PROGRAM EventLog


VAR
	WriteTest		:	BOOL;
	fbOpenFile 		: FB_Fileopen;
	fbWriteFile		: FB_FilePuts;
	fbCloseFile 	: FB_FileClose;
	fbRenameFile	: FB_FileRename;
	fbDeleteFile	: FB_FileDelete;
	fbFileInfo		:	FB_EnumFindFileEntry;
	stFiledata		:	ST_FindFileEntry;
	FileOpenDone		:	F_TRIG;
	FileWriteDone		:	F_TRIG;
	FileCloseDone		:	F_TRIG;
	FileRenameDone		:	F_TRIG;
	FileDeleteDone		:	F_TRIG;
	FileInfoDone		:	F_TRIG;
	FileSize			:	ULINT;
	FileCounter			:	INT;
	Filehandle 			: UINT;
	
	bForceWrite 			:	BOOL;	//immediately flush out buffer on shutdown
	bEMstopWrite			:	BOOL;	//Flush out after EMStop, but give some time for final logs to come in 
	tonEMstopDelay			:	TON;
	tonGeneralWriteDelay	:	Ton;
	FileActionDelay			:	TON := (PT := T#30MS);

	MemoryBuffer	:	FB_StringRingBuffer;
	DataBuffer		:	ARRAY[0..100000] OF BYTE; //100kb to start
	WriteString	:	t_MAXSTRING;

	
	
	Stop_logging	:	Bool;
	
END_VAR

VAR_IN_OUT CONSTANT
	STParams : ST_EventLoggerParams;
END_VAR

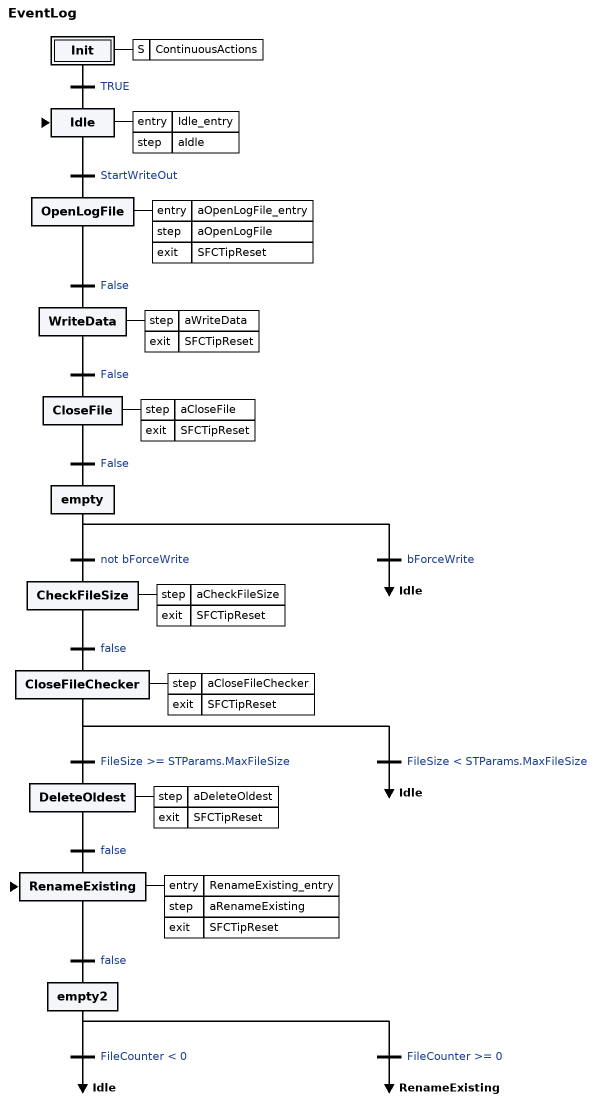
INITIAL_STEP Init:
    ContinuousActions(S);
END_STEP
TRANSITION FROM Init TO Idle
    := TRUE;
END_TRANSITION
STEP Idle:
    Idle_entry(P1);  // entry action
    aIdle(N);  // step action
END_STEP
TRANSITION FROM Idle TO OpenLogFile
    := StartWriteOut;
END_TRANSITION
// macro Writeout begins
STEP OpenLogFile:
    aOpenLogFile_entry(P1);  // entry action
    aOpenLogFile(N);  // step action
    SFCTipReset(P0);  // exit action
END_STEP
TRANSITION FROM OpenLogFile TO WriteData
    := False;
END_TRANSITION
STEP WriteData:
    aWriteData(N);  // step action
    SFCTipReset(P0);  // exit action
END_STEP
TRANSITION FROM WriteData TO CloseFile
    := False;
END_TRANSITION
STEP CloseFile:
    aCloseFile(N);  // step action
    SFCTipReset(P0);  // exit action
END_STEP
TRANSITION FROM CloseFile TO empty
    := False;
END_TRANSITION
STEP empty:
END_STEP
TRANSITION FROM empty TO CheckFileSize
    := not bForceWrite;
END_TRANSITION
TRANSITION FROM empty TO Idle
    := bForceWrite;
END_TRANSITION
// macro LogRotate begins
STEP CheckFileSize:
    aCheckFileSize(N);  // step action
    SFCTipReset(P0);  // exit action
END_STEP
TRANSITION FROM CheckFileSize TO CloseFileChecker
    := false;
END_TRANSITION
STEP CloseFileChecker:
    aCloseFileChecker(N);  // step action
    SFCTipReset(P0);  // exit action
END_STEP
TRANSITION FROM CloseFileChecker TO DeleteOldest
    := FileSize >= STParams.MaxFileSize;
END_TRANSITION
STEP DeleteOldest:
    aDeleteOldest(N);  // step action
    SFCTipReset(P0);  // exit action
END_STEP
TRANSITION FROM DeleteOldest TO RenameExisting
    := false;
END_TRANSITION
STEP RenameExisting:
    RenameExisting_entry(P1);  // entry action
    aRenameExisting(N);  // step action
    SFCTipReset(P0);  // exit action
END_STEP
TRANSITION FROM RenameExisting TO empty2
    := false;
END_TRANSITION
STEP empty2:
END_STEP
TRANSITION FROM empty2 TO Idle
    := FileCounter < 0;
END_TRANSITION
TRANSITION FROM empty2 TO RenameExisting
    := FileCounter >= 0;
END_TRANSITION
TRANSITION FROM CloseFileChecker TO Idle
    := FileSize < STParams.MaxFileSize;
END_TRANSITION

ACTION aCheckFileSize:


FileInfoDone(clk := fbFileInfo.bbusy);
FileActionDelay(in:= NOT (fbFileInfo.bbusy OR FileInfoDone.Q));

fbFileInfo(sPathname:= Stparams.LogFileName,
		bExecute := FileActionDelay.Q,
		eCMD := eEnumCmd_First,
		tTimeout := T#100MS);


IF FileInfoDone.q THEN
	FileSize := 0;
	IF NOT fbFileInfo.bError THEN
		IF NOT fbfileInfo.bEOE THEN
			stFiledata := fbFileinfo.stFindFile;
			FileSize := ULARGE_TO_ULINT(stFiledata.fileSize);
		END_IF
	END_IF
	SFCTip := TRUE;
END_IF
END_ACTION

ACTION aCloseFile:

FileCloseDone(clk := fbCloseFile.bbusy);

FileActionDelay(in := NOT (fbCloseFile.bbusy OR FileCloseDone.Q));


fbCloseFile(Hfile := FileHandle,
		bExecute   := FileActionDelay.q,
    	tTimeout   := T#100MS);


IF FileCloseDone.q THEN
	IF NOT fbCloseFile.bError THEN
		filehandle := 0;
		SFCTip := TRUE;
	END_IF
END_IF
END_ACTION

ACTION aCloseFileChecker:


FileInfoDone(clk := fbFileInfo.bbusy);
FileActionDelay(in:= not (fbFileInfo.bbusy OR FileInfoDone.Q));

fbFileInfo(sPathname:= Stparams.LogFileName,
		bExecute := FileActionDelay.Q,
		eCMD := eEnumCmd_Abort,
		tTimeout := T#100MS);


IF FileInfoDone.q THEN
	FileSize := 0;
	IF NOT fbFileInfo.bError THEN
		SFCTip := TRUE;
	END_IF
END_IF
END_ACTION

METHOD AddEvent : BOOL
VAR_INPUT
	LogMessage	:	STRING;
END_VAR
IF NOT Stop_logging THEN	
	MemoryBuffer.A_AddTail(putValue := LogMessage);
end_if
END_METHOD

ACTION aDeleteOldest:

FileDeleteDone(clk := fbDeleteFile.bbusy);
FileActionDelay(in:=NOT (fbDeleteFile.bbusy OR FileDeleteDone.Q));
	
fbDeleteFile(sPathname:= concat(concat(Stparams.LogFileName, '.'),TO_STRING(stparams.MaxFileCount-1)),
		bExecute := FileActionDelay.q,
		tTimeout := T#100MS);


IF FileDeleteDone.q THEN
	//could end in error if file doesn't exist. This is fine.
	FileCounter := stparams.MaxFileCount-2;
	SFCTip := TRUE;
END_IF
END_ACTION

ACTION aIdle:
tonGeneralWriteDelay.IN := true;
END_ACTION

ACTION aOpenLogFile:
bEMStopWrite := FALSE;
tonGeneralWriteDelay.IN := FALSE;
FileOpenDone(clk := fbOpenFile.bbusy);

FileActionDelay(in := NOT (fbOpenFile.bbusy OR FileOpenDone.Q));

fbOpenFile(sPathName := Stparams.LogFileName,
		nMode := FOPEN_MODEAPPEND OR FOPEN_MODETEXT,
		bExecute   :=  FileActionDelay.Q,
    	tTimeout   := T#100MS);


IF FileOpenDone.q THEN
	FileHandle := fbOpenFile.hFile;
	IF FileHandle <> 0 THEN
		MemoryBuffer.A_RemoveHead(getValue => WriteString);
		SFCTip := TRUE;
	END_IF
END_IF
END_ACTION

ACTION aOpenLogFile_entry:

END_ACTION

ACTION aRenameExisting:

FileRenameDone(clk := fbRenameFile.bbusy);
FileActionDelay(in:= NOT (fbDeleteFile.bbusy OR FileDeleteDone.Q));

fbRenameFile(
		bExecute := FileActionDelay.Q,
		tTimeout := T#100MS);


IF FileRenameDone.q THEN
	//could end in error if file doesn't exist. This is fine.
	FileCounter := FileCounter-1;
	SFCTip := TRUE;
END_IF
END_ACTION

ACTION aWriteData:

//add entry action with initial Writestring fill
filehandle;

FileWriteDone(clk := fbWriteFile.bbusy);

FileActionDelay(in := NOT (fbWriteFile.bbusy OR FileWriteDone.Q));

fbWriteFile(hfile := filehandle,
			sLine := WriteString,
			BExecute := FileActionDelay.Q,
			tTimeout := T#500MS);


IF FileWriteDone.q THEN
	IF MemoryBuffer.nCount > 0 THEN //Still data present, continue writing
		MemoryBuffer.A_RemoveHead(getValue => WriteString);
	ELSE //file not opened, back to start?
		SFCTip := TRUE;
	END_IF
END_IF
END_ACTION

ACTION ContinuousActions:
MemoryBuffer(bOverwrite := TRUE, pBuffer := ADR(DataBuffer), cbBuffer := SIZEOF(DataBuffer));
tonEMstopDelay(in := bEMstopWrite, pt:= stparams.EMstopWriteDelay);
tonGeneralWriteDelay(in:= MemoryBuffer.nCount > 0, Pt:=stparams.LogWriteInterval);

IF WriteTest THEN
	WriteLogItem(Source := eObject_ID.System, Severity := eSeverity.Warning, LogText := 'testtesttest');
	WriteTest := FALSE;
	bEMstopWrite := TRUE;
END_IF
END_ACTION

METHOD EMstop : BOOL
VAR_INPUT
END_VAR

VAR
	LogText	:	String;
END_VAR

IF memorybuffer.nCount > 0 THEN
	bEMstopWrite := TRUE;
END_IF

EMStop := TRUE;
END_METHOD

ACTION Idle_entry:
bEMStopWrite := FALSE;
bForceWrite := FALSE;
END_ACTION

ACTION RenameExisting_entry:

IF FileCounter = 0 THEN 
	fbRenameFile.sOldName := Stparams.LogFileName;
ELSE
	fbRenameFile.sOldName := concat(concat(Stparams.LogFileName, '.'),TO_STRING(FileCounter));
END_IF
fbRenameFile.sNewName	:= concat(concat(Stparams.LogFileName, '.'),TO_STRING(FileCounter+1));
END_ACTION

ACTION SFCTipReset:
FileActionDelay(in := FALSE);
SFCTip := false;
END_ACTION

METHOD Shutdown : BOOL
VAR_INPUT
END_VAR

IF memorybuffer.nCount > 0 THEN
	bForceWrite := TRUE;
END_IF

Shutdown := TRUE;
END_METHOD

TRANSITION StartWriteOut:
//Flush logs to file if
MemoryBuffer.cbSize > TO_UDINT(stparams.MaxFillGrade*MemoryBuffer.cbBuffer) OR //buffer gets full
tonGeneralWriteDelay.Q  OR //fixed interval
tonEmstopDelay.Q OR //just after emstop
bForceWrite; //at systemshutdown
END_TRANSITION

END_PROGRAM

(* stored: Version 1.1.0.1, ProductVersion 3.1.4024.12
   POU EventLog: Id {9182a965-c0a3-47fb-8d9e-fc3986a324a0}, SpecialFunc None
   Folder private: Id {39773113-d3ca-4aed-b4c6-9841f9e50aea}
   Action aCheckFileSize: Id {58585cd0-1a18-4507-ae00-a1805d81c4ea}
   Action aCloseFile: Id {ea5efb7d-ae55-4798-83dd-00d5a01807ec}
   Action aCloseFileChecker: Id {cffd68e5-23a5-4609-90f6-a609898df913}
   Method AddEvent: Id {32cb5227-5b76-4542-a4a3-ceb6eedbd564}
   Action aDeleteOldest: Id {3e17bcae-26df-43ff-b063-d7004346f315}
   Action aIdle: Id {30d500f2-9720-4731-a0c6-2f3df7932a4e}
   Action aOpenLogFile: Id {cb185fb2-912d-4e72-b610-3cad69402948}
   Action aOpenLogFile_entry: Id {d319d2ef-8988-4c8d-bad7-a84e46814636}
   Action aRenameExisting: Id {73354ae8-5d50-4c42-ab51-78b56e0ea2e3}
   Action aWriteData: Id {a30c5a53-376d-4075-ad71-90040a3b5b86}
   Action ContinuousActions: Id {6ab03acc-c81e-4be5-914d-eb93b7fac4cc}
   Method EMstop: Id {2864481c-1419-4b09-8c6e-efbb21d146a6}
   Action Idle_entry: Id {d5f7fac5-8387-4d6f-be5f-57dfbc81f95a}
   Action RenameExisting_entry: Id {6f3681b5-e206-409f-bc97-e8cdd8d50fb1}
   Action SFCTipReset: Id {1162c354-8e0f-41e9-b76e-d82acb041b53}
   Method Shutdown: Id {66d78e64-779f-4597-a532-ba74365e3190}
   Transition StartWriteOut: Id {f3d5451a-7330-4920-99a0-9c375ad1e788} *)
